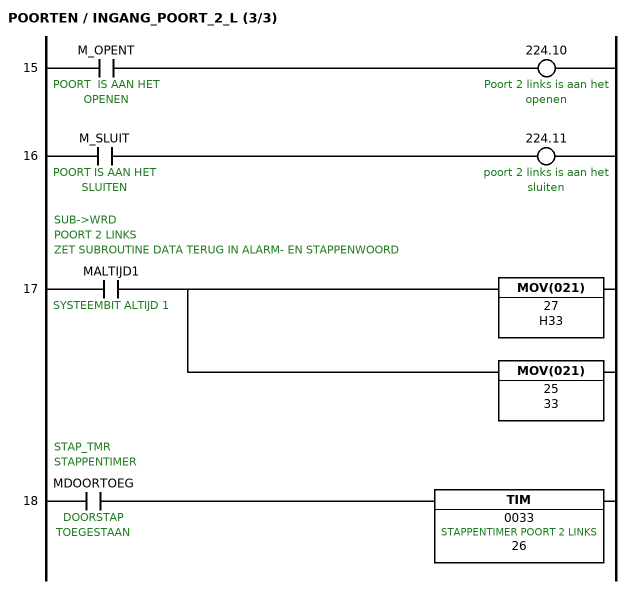
; [picture p445: POORTEN / INGANG_POORT_2_L, rungs 15-18]
; rung 15
LD M_OPENT  ; POORT  IS AAN HET OPENEN
OUT 224.10  ; Poort 2 links is aan het openen
; rung 16
LD M_SLUIT  ; POORT IS AAN HET SLUITEN
OUT 224.11  ; poort 2 links is aan het sluiten
; rung 17: SUB->WRD / POORT 2 LINKS / ZET SUBROUTINE DATA TERUG IN ALARM- EN STAPPENWOORD
LD MALTIJD1  ; SYSTEEMBIT ALTIJD 1
MOV(021) 27 H33
MOV(021) 25 33
; rung 18: STAP_TMR / STAPPENTIMER
LD MDOORTOEG  ; DOORSTAP TOEGESTAAN
TIM 0033 26  ; STAPPENTIMER POORT 2 LINKS

### Section INGANG_POORT_2_R

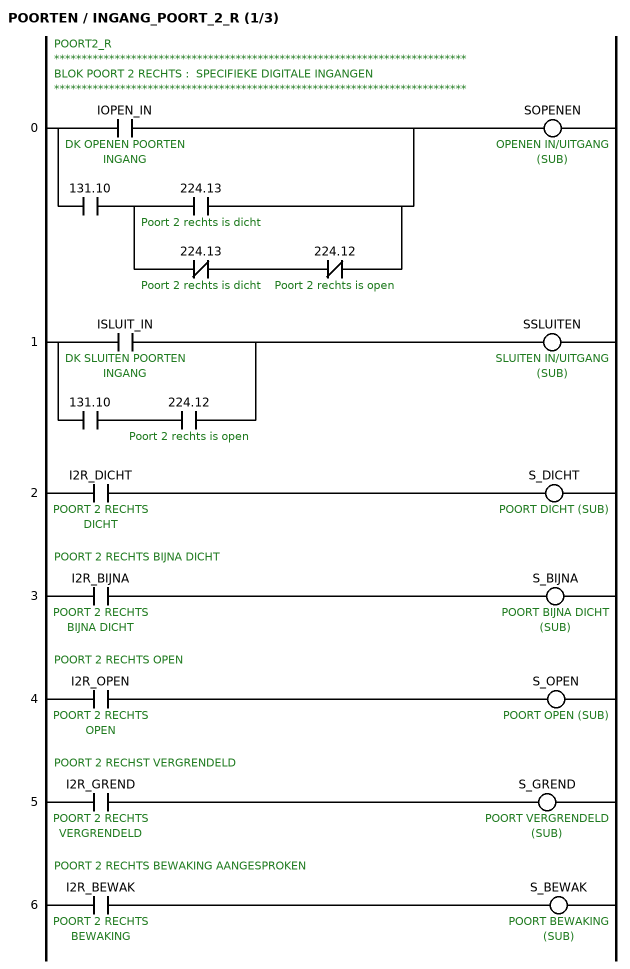
; rung 0: POORT2_R / *************************************************************************** / BLOK POORT 2 RECHTS :  SPECIFIEKE DIGITALE INGANGEN / ***************************************************************************
LD IOPEN_IN  ; DK OPENEN POORTEN INGANG
LD 131.10
LD 224.13  ; Poort 2 rechts is dicht
LDNOT 224.13  ; Poort 2 rechts is dicht
ANDNOT 224.12  ; Poort 2 rechts is open
ORLD
ANDLD
ORLD
OUT SOPENEN  ; OPENEN IN/UITGANG (SUB)
; rung 1
LD ISLUIT_IN  ; DK SLUITEN POORTEN INGANG
LD 131.10
AND 224.12  ; Poort 2 rechts is open
ORLD
OUT SSLUITEN  ; SLUITEN IN/UITGANG (SUB)
; rung 2
LD I2R_DICHT  ; POORT 2 RECHTS DICHT
OUT S_DICHT  ; POORT DICHT (SUB)
; rung 3: POORT 2 RECHTS BIJNA DICHT
LD I2R_BIJNA  ; POORT 2 RECHTS BIJNA DICHT
OUT S_BIJNA  ; POORT BIJNA DICHT (SUB)
; rung 4: POORT 2 RECHTS OPEN
LD I2R_OPEN  ; POORT 2 RECHTS OPEN
OUT S_OPEN  ; POORT OPEN (SUB)
; rung 5: POORT 2 RECHST VERGRENDELD
LD I2R_GREND  ; POORT 2 RECHTS VERGRENDELD
OUT S_GREND  ; POORT VERGRENDELD  (SUB)
; rung 6: POORT 2 RECHTS BEWAKING AANGESPROKEN
LD I2R_BEWAK  ; POORT 2 RECHTS BEWAKING
OUT S_BEWAK  ; POORT BEWAKING  (SUB)

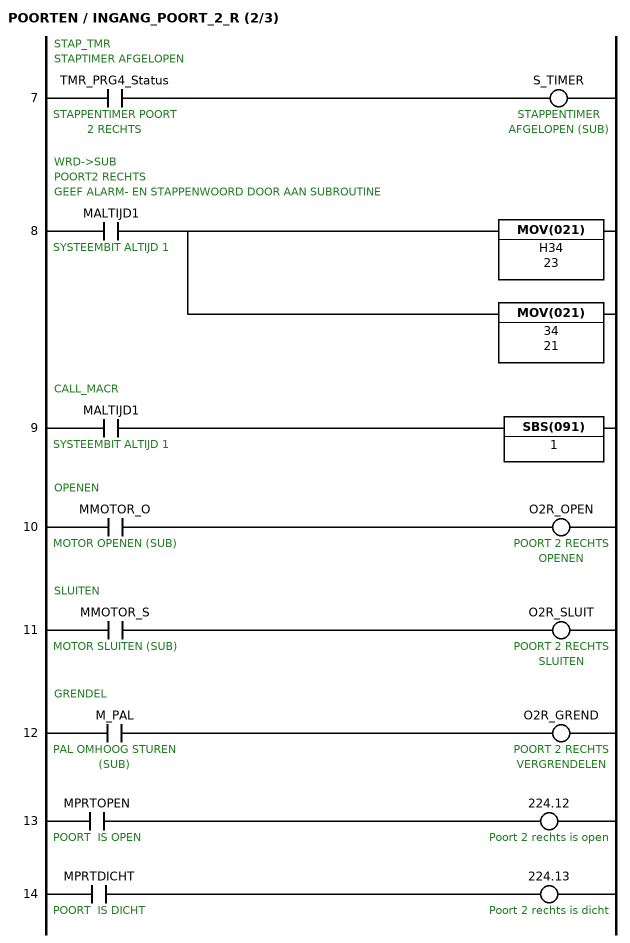
; rung 7: STAP_TMR / STAPTIMER AFGELOPEN
LD TMR_PRG4_Status  ; STAPPENTIMER POORT 2 RECHTS
OUT S_TIMER  ; STAPPENTIMER AFGELOPEN (SUB)
; rung 8: WRD->SUB / POORT2 RECHTS / GEEF ALARM- EN STAPPENWOORD DOOR AAN SUBROUTINE
LD MALTIJD1  ; SYSTEEMBIT ALTIJD 1
MOV(021) H34 23
MOV(021) 34 21
; rung 9: CALL_MACR
LD MALTIJD1  ; SYSTEEMBIT ALTIJD 1
SBS(091) 1
; rung 10: OPENEN
LD MMOTOR_O  ; MOTOR OPENEN (SUB)
OUT O2R_OPEN  ; POORT 2 RECHTS OPENEN
; rung 11: SLUITEN
LD MMOTOR_S  ; MOTOR SLUITEN (SUB)
OUT O2R_SLUIT  ; POORT 2 RECHTS SLUITEN
; rung 12: GRENDEL
LD M_PAL  ; PAL OMHOOG STUREN (SUB)
OUT O2R_GREND  ; POORT 2 RECHTS VERGRENDELEN
; rung 13
LD MPRTOPEN  ; POORT  IS OPEN
OUT 224.12  ; Poort 2 rechts is open
; rung 14
LD MPRTDICHT  ; POORT  IS DICHT
OUT 224.13  ; Poort 2 rechts is dicht

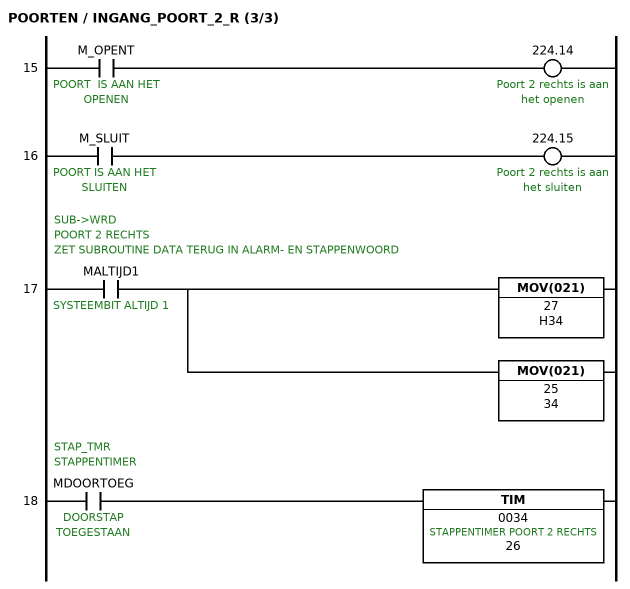
; rung 15
LD M_OPENT  ; POORT  IS AAN HET OPENEN
OUT 224.14  ; Poort 2 rechts is aan het openen
; rung 16
LD M_SLUIT  ; POORT IS AAN HET SLUITEN
OUT 224.15  ; Poort 2 rechts is aan het sluiten
; rung 17: SUB->WRD / POORT 2 RECHTS / ZET SUBROUTINE DATA TERUG IN ALARM- EN STAPPENWOORD
LD MALTIJD1  ; SYSTEEMBIT ALTIJD 1
MOV(021) 27 H34
MOV(021) 25 34
; rung 18: STAP_TMR / STAPPENTIMER
LD MDOORTOEG  ; DOORSTAP TOEGESTAAN
TIM 0034 26  ; STAPPENTIMER POORT 2 RECHTS

### Section UITGANG_POORT_3_L

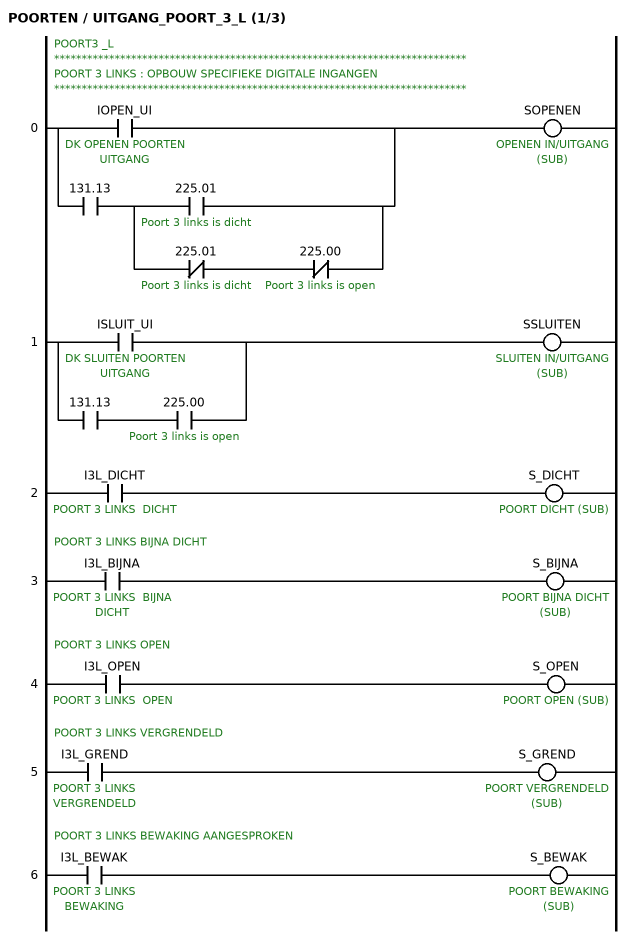
; rung 0: POORT3 _L / *************************************************************************** / POORT 3 LINKS : OPBOUW SPECIFIEKE DIGITALE INGANGEN / ***************************************************************************
LD IOPEN_UI  ; DK OPENEN POORTEN UITGANG
LD 131.13
LD 225.01  ; Poort 3 links is dicht
LDNOT 225.01  ; Poort 3 links is dicht
ANDNOT 225.00  ; Poort 3 links is open
ORLD
ANDLD
ORLD
OUT SOPENEN  ; OPENEN IN/UITGANG (SUB)
; rung 1
LD ISLUIT_UI  ; DK SLUITEN POORTEN UITGANG
LD 131.13
AND 225.00  ; Poort 3 links is open
ORLD
OUT SSLUITEN  ; SLUITEN IN/UITGANG (SUB)
; rung 2
LD I3L_DICHT  ; POORT 3 LINKS  DICHT
OUT S_DICHT  ; POORT DICHT (SUB)
; rung 3: POORT 3 LINKS BIJNA DICHT
LD I3L_BIJNA  ; POORT 3 LINKS  BIJNA DICHT
OUT S_BIJNA  ; POORT BIJNA DICHT (SUB)
; rung 4: POORT 3 LINKS OPEN
LD I3L_OPEN  ; POORT 3 LINKS  OPEN
OUT S_OPEN  ; POORT OPEN (SUB)
; rung 5: POORT 3 LINKS VERGRENDELD
LD I3L_GREND  ; POORT 3 LINKS VERGRENDELD
OUT S_GREND  ; POORT VERGRENDELD  (SUB)
; rung 6: POORT 3 LINKS BEWAKING AANGESPROKEN
LD I3L_BEWAK  ; POORT 3 LINKS BEWAKING
OUT S_BEWAK  ; POORT BEWAKING  (SUB)

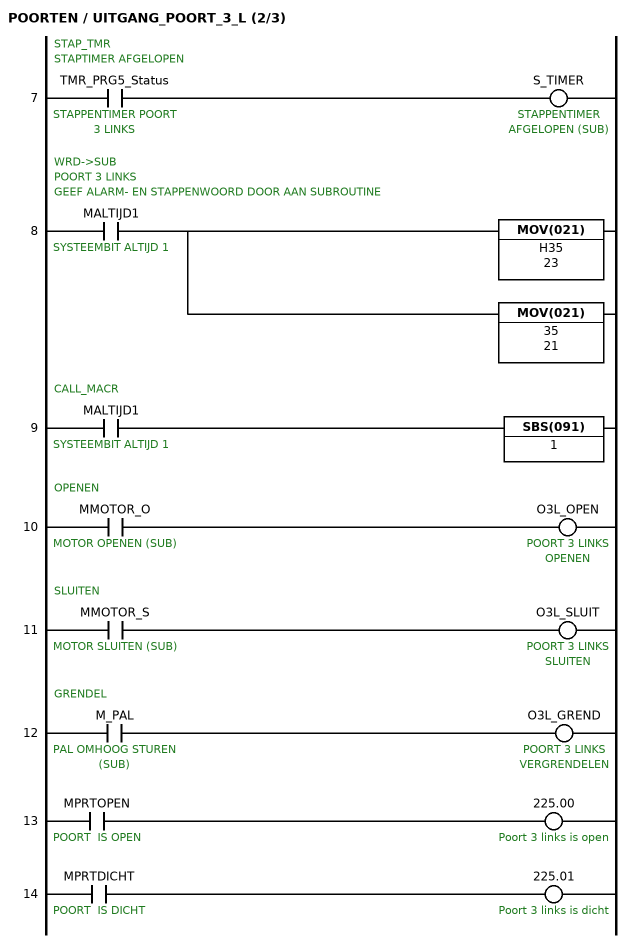
; rung 7: STAP_TMR / STAPTIMER AFGELOPEN
LD TMR_PRG5_Status  ; STAPPENTIMER POORT 3 LINKS
OUT S_TIMER  ; STAPPENTIMER AFGELOPEN (SUB)
; rung 8: WRD->SUB / POORT 3 LINKS / GEEF ALARM- EN STAPPENWOORD DOOR AAN SUBROUTINE
LD MALTIJD1  ; SYSTEEMBIT ALTIJD 1
MOV(021) H35 23
MOV(021) 35 21
; rung 9: CALL_MACR
LD MALTIJD1  ; SYSTEEMBIT ALTIJD 1
SBS(091) 1
; rung 10: OPENEN
LD MMOTOR_O  ; MOTOR OPENEN (SUB)
OUT O3L_OPEN  ; POORT 3 LINKS OPENEN
; rung 11: SLUITEN
LD MMOTOR_S  ; MOTOR SLUITEN (SUB)
OUT O3L_SLUIT  ; POORT 3 LINKS SLUITEN
; rung 12: GRENDEL
LD M_PAL  ; PAL OMHOOG STUREN (SUB)
OUT O3L_GREND  ; POORT 3 LINKS VERGRENDELEN
; rung 13
LD MPRTOPEN  ; POORT  IS OPEN
OUT 225.00  ; Poort 3 links is open
; rung 14
LD MPRTDICHT  ; POORT  IS DICHT
OUT 225.01  ; Poort 3 links is dicht

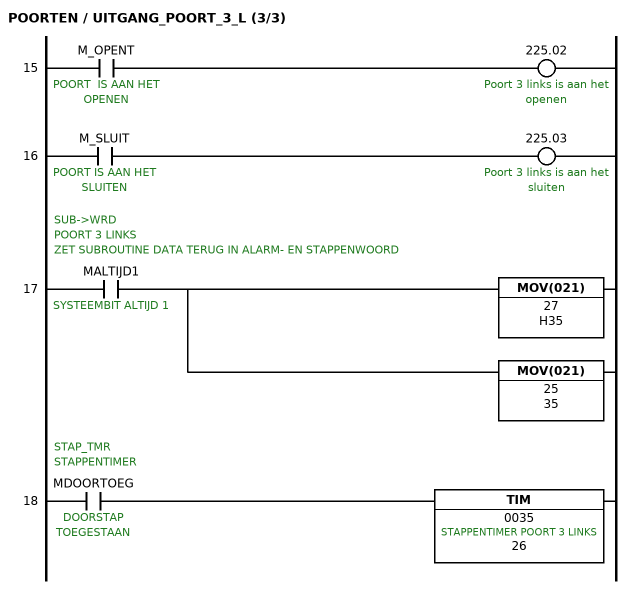
; rung 15
LD M_OPENT  ; POORT  IS AAN HET OPENEN
OUT 225.02  ; Poort 3 links is aan het openen
; rung 16
LD M_SLUIT  ; POORT IS AAN HET SLUITEN
OUT 225.03  ; Poort 3 links is aan het sluiten
; rung 17: SUB->WRD / POORT 3 LINKS / ZET SUBROUTINE DATA TERUG IN ALARM- EN STAPPENWOORD
LD MALTIJD1  ; SYSTEEMBIT ALTIJD 1
MOV(021) 27 H35
MOV(021) 25 35
; rung 18: STAP_TMR / STAPPENTIMER
LD MDOORTOEG  ; DOORSTAP TOEGESTAAN
TIM 0035 26  ; STAPPENTIMER POORT 3 LINKS

### Section UITGANG_POORT_3_R

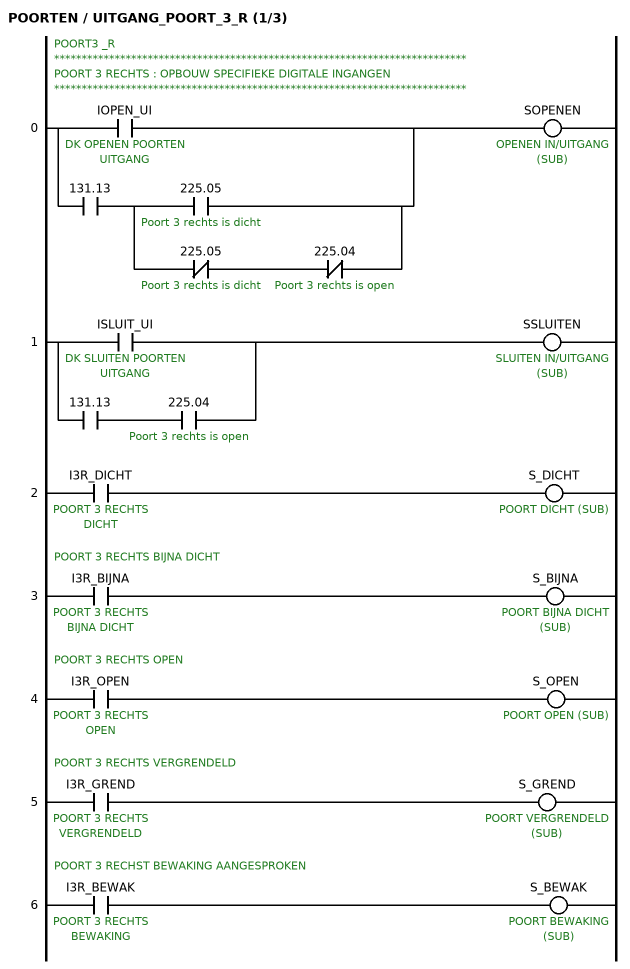
; rung 0: POORT3 _R / *************************************************************************** / POORT 3 RECHTS : OPBOUW SPECIFIEKE DIGITALE INGANGEN / ***************************************************************************
LD IOPEN_UI  ; DK OPENEN POORTEN UITGANG
LD 131.13
LD 225.05  ; Poort 3 rechts is dicht
LDNOT 225.05  ; Poort 3 rechts is dicht
ANDNOT 225.04  ; Poort 3 rechts is open
ORLD
ANDLD
ORLD
OUT SOPENEN  ; OPENEN IN/UITGANG (SUB)
; rung 1
LD ISLUIT_UI  ; DK SLUITEN POORTEN UITGANG
LD 131.13
AND 225.04  ; Poort 3 rechts is open
ORLD
OUT SSLUITEN  ; SLUITEN IN/UITGANG (SUB)
; rung 2
LD I3R_DICHT  ; POORT 3 RECHTS DICHT
OUT S_DICHT  ; POORT DICHT (SUB)
; rung 3: POORT 3 RECHTS BIJNA DICHT
LD I3R_BIJNA  ; POORT 3 RECHTS BIJNA DICHT
OUT S_BIJNA  ; POORT BIJNA DICHT (SUB)
; rung 4: POORT 3 RECHTS OPEN
LD I3R_OPEN  ; POORT 3 RECHTS OPEN
OUT S_OPEN  ; POORT OPEN (SUB)
; rung 5: POORT 3 RECHTS VERGRENDELD
LD I3R_GREND  ; POORT 3 RECHTS VERGRENDELD
OUT S_GREND  ; POORT VERGRENDELD  (SUB)
; rung 6: POORT 3 RECHST BEWAKING AANGESPROKEN
LD I3R_BEWAK  ; POORT 3 RECHTS BEWAKING
OUT S_BEWAK  ; POORT BEWAKING  (SUB)

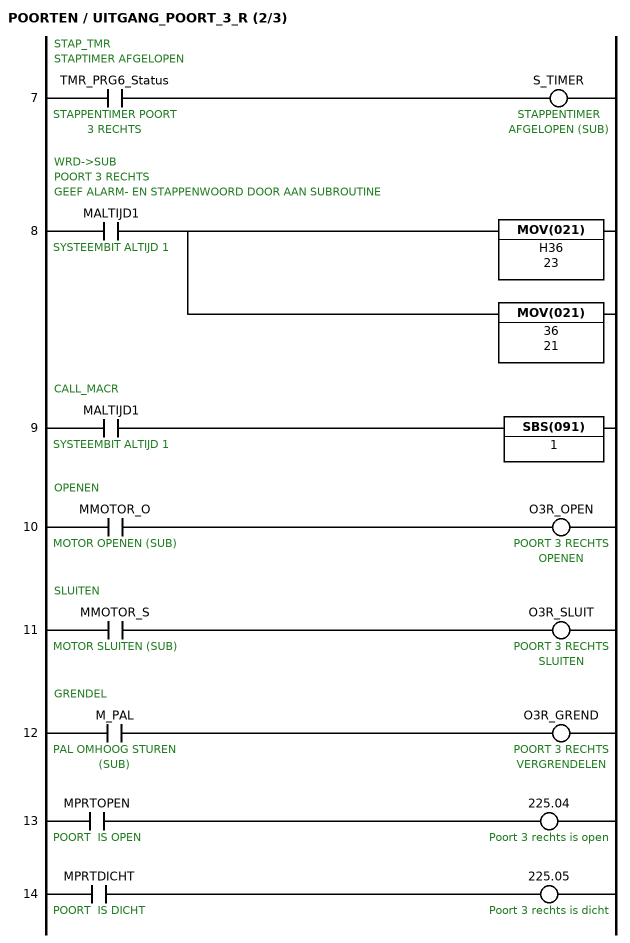
; rung 7: STAP_TMR / STAPTIMER AFGELOPEN
LD TMR_PRG6_Status  ; STAPPENTIMER POORT 3 RECHTS
OUT S_TIMER  ; STAPPENTIMER AFGELOPEN (SUB)
; rung 8: WRD->SUB / POORT 3 RECHTS / GEEF ALARM- EN STAPPENWOORD DOOR AAN SUBROUTINE
LD MALTIJD1  ; SYSTEEMBIT ALTIJD 1
MOV(021) H36 23
MOV(021) 36 21
; rung 9: CALL_MACR
LD MALTIJD1  ; SYSTEEMBIT ALTIJD 1
SBS(091) 1
; rung 10: OPENEN
LD MMOTOR_O  ; MOTOR OPENEN (SUB)
OUT O3R_OPEN  ; POORT 3 RECHTS OPENEN
; rung 11: SLUITEN
LD MMOTOR_S  ; MOTOR SLUITEN (SUB)
OUT O3R_SLUIT  ; POORT 3 RECHTS SLUITEN
; rung 12: GRENDEL
LD M_PAL  ; PAL OMHOOG STUREN (SUB)
OUT O3R_GREND  ; POORT 3 RECHTS VERGRENDELEN
; rung 13
LD MPRTOPEN  ; POORT  IS OPEN
OUT 225.04  ; Poort 3 rechts is open
; rung 14
LD MPRTDICHT  ; POORT  IS DICHT
OUT 225.05  ; Poort 3 rechts is dicht

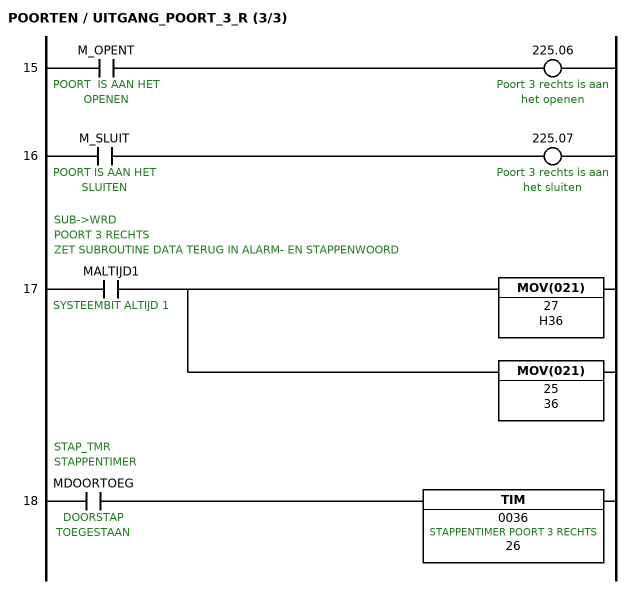
; rung 15
LD M_OPENT  ; POORT  IS AAN HET OPENEN
OUT 225.06  ; Poort 3 rechts is aan het openen
; rung 16
LD M_SLUIT  ; POORT IS AAN HET SLUITEN
OUT 225.07  ; Poort 3 rechts is aan het sluiten
; rung 17: SUB->WRD / POORT 3 RECHTS / ZET SUBROUTINE DATA TERUG IN ALARM- EN STAPPENWOORD
LD MALTIJD1  ; SYSTEEMBIT ALTIJD 1
MOV(021) 27 H36
MOV(021) 25 36
; rung 18: STAP_TMR / STAPPENTIMER
LD MDOORTOEG  ; DOORSTAP TOEGESTAAN
TIM 0036 26  ; STAPPENTIMER POORT 3 RECHTS

### Section UITGANG_POORT_4_L

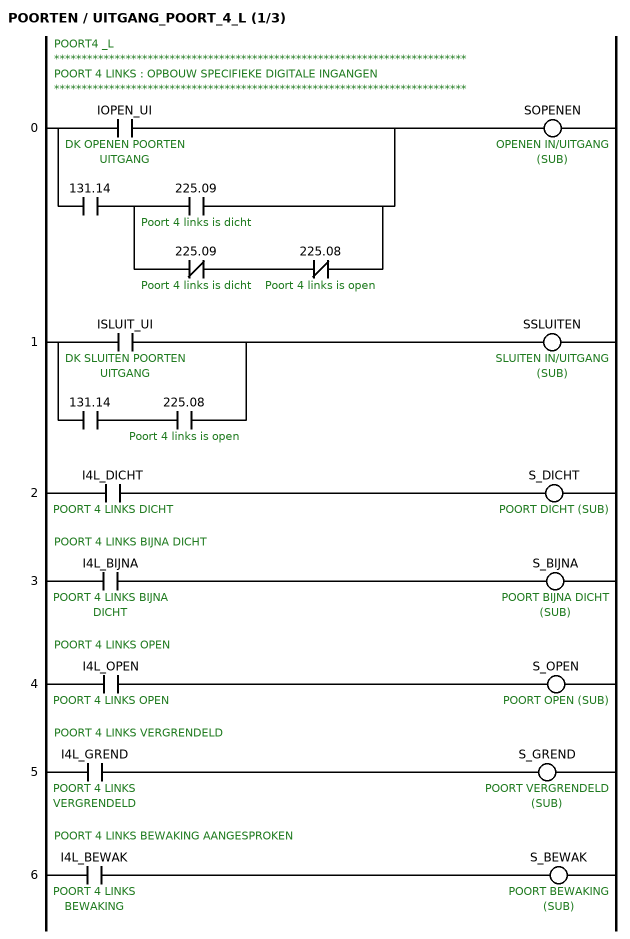
; rung 0: POORT4 _L / *************************************************************************** / POORT 4 LINKS : OPBOUW SPECIFIEKE DIGITALE INGANGEN / ***************************************************************************
LD IOPEN_UI  ; DK OPENEN POORTEN UITGANG
LD 131.14
LD 225.09  ; Poort 4 links is dicht
LDNOT 225.09  ; Poort 4 links is dicht
ANDNOT 225.08  ; Poort 4 links is open
ORLD
ANDLD
ORLD
OUT SOPENEN  ; OPENEN IN/UITGANG (SUB)
; rung 1
LD ISLUIT_UI  ; DK SLUITEN POORTEN UITGANG
LD 131.14
AND 225.08  ; Poort 4 links is open
ORLD
OUT SSLUITEN  ; SLUITEN IN/UITGANG (SUB)
; rung 2
LD I4L_DICHT  ; POORT 4 LINKS DICHT
OUT S_DICHT  ; POORT DICHT (SUB)
; rung 3: POORT 4 LINKS BIJNA DICHT
LD I4L_BIJNA  ; POORT 4 LINKS BIJNA DICHT
OUT S_BIJNA  ; POORT BIJNA DICHT (SUB)
; rung 4: POORT 4 LINKS OPEN
LD I4L_OPEN  ; POORT 4 LINKS OPEN
OUT S_OPEN  ; POORT OPEN (SUB)
; rung 5: POORT 4 LINKS VERGRENDELD
LD I4L_GREND  ; POORT 4 LINKS VERGRENDELD
OUT S_GREND  ; POORT VERGRENDELD  (SUB)
; rung 6: POORT 4 LINKS BEWAKING AANGESPROKEN
LD I4L_BEWAK  ; POORT 4 LINKS BEWAKING
OUT S_BEWAK  ; POORT BEWAKING  (SUB)

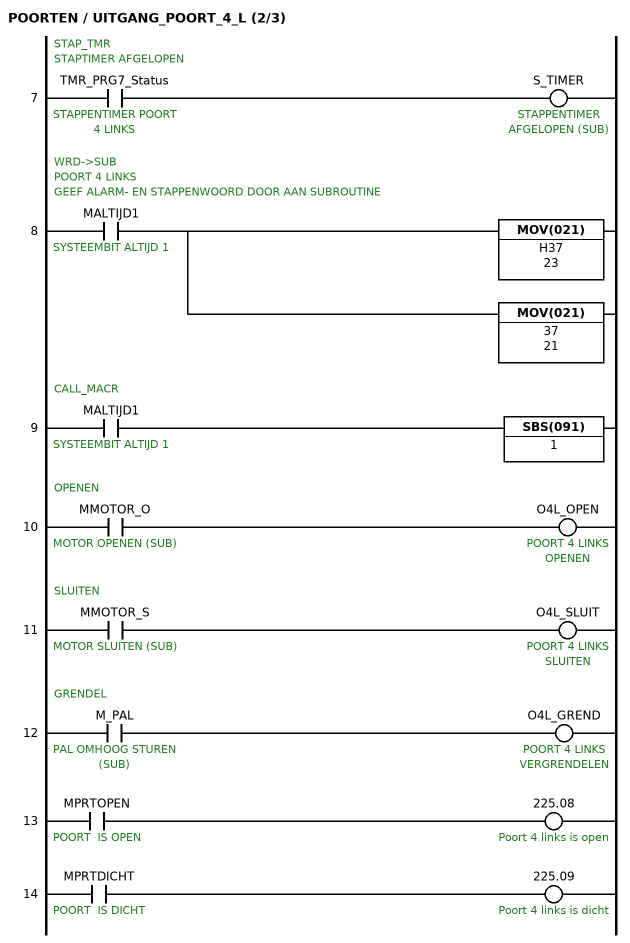
; rung 7: STAP_TMR / STAPTIMER AFGELOPEN
LD TMR_PRG7_Status  ; STAPPENTIMER POORT 4 LINKS
OUT S_TIMER  ; STAPPENTIMER AFGELOPEN (SUB)
; rung 8: WRD->SUB / POORT 4 LINKS / GEEF ALARM- EN STAPPENWOORD DOOR AAN SUBROUTINE
LD MALTIJD1  ; SYSTEEMBIT ALTIJD 1
MOV(021) H37 23
MOV(021) 37 21
; rung 9: CALL_MACR
LD MALTIJD1  ; SYSTEEMBIT ALTIJD 1
SBS(091) 1
; rung 10: OPENEN
LD MMOTOR_O  ; MOTOR OPENEN (SUB)
OUT O4L_OPEN  ; POORT 4 LINKS OPENEN
; rung 11: SLUITEN
LD MMOTOR_S  ; MOTOR SLUITEN (SUB)
OUT O4L_SLUIT  ; POORT 4 LINKS SLUITEN
; rung 12: GRENDEL
LD M_PAL  ; PAL OMHOOG STUREN (SUB)
OUT O4L_GREND  ; POORT 4 LINKS VERGRENDELEN
; rung 13
LD MPRTOPEN  ; POORT  IS OPEN
OUT 225.08  ; Poort 4 links is open
; rung 14
LD MPRTDICHT  ; POORT  IS DICHT
OUT 225.09  ; Poort 4 links is dicht

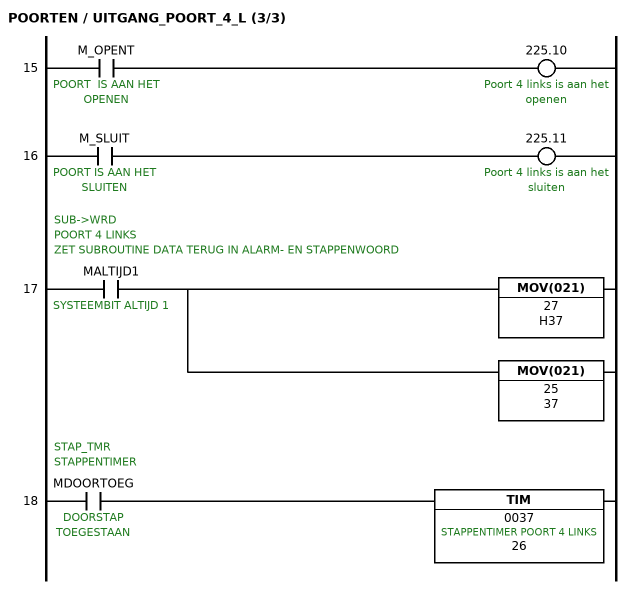
; rung 15
LD M_OPENT  ; POORT  IS AAN HET OPENEN
OUT 225.10  ; Poort 4 links is aan het openen
; rung 16
LD M_SLUIT  ; POORT IS AAN HET SLUITEN
OUT 225.11  ; Poort 4 links is aan het sluiten
; rung 17: SUB->WRD / POORT 4 LINKS / ZET SUBROUTINE DATA TERUG IN ALARM- EN STAPPENWOORD
LD MALTIJD1  ; SYSTEEMBIT ALTIJD 1
MOV(021) 27 H37
MOV(021) 25 37
; rung 18: STAP_TMR / STAPPENTIMER
LD MDOORTOEG  ; DOORSTAP TOEGESTAAN
TIM 0037 26  ; STAPPENTIMER POORT 4 LINKS

### Section UITGANG_POORT_4_R

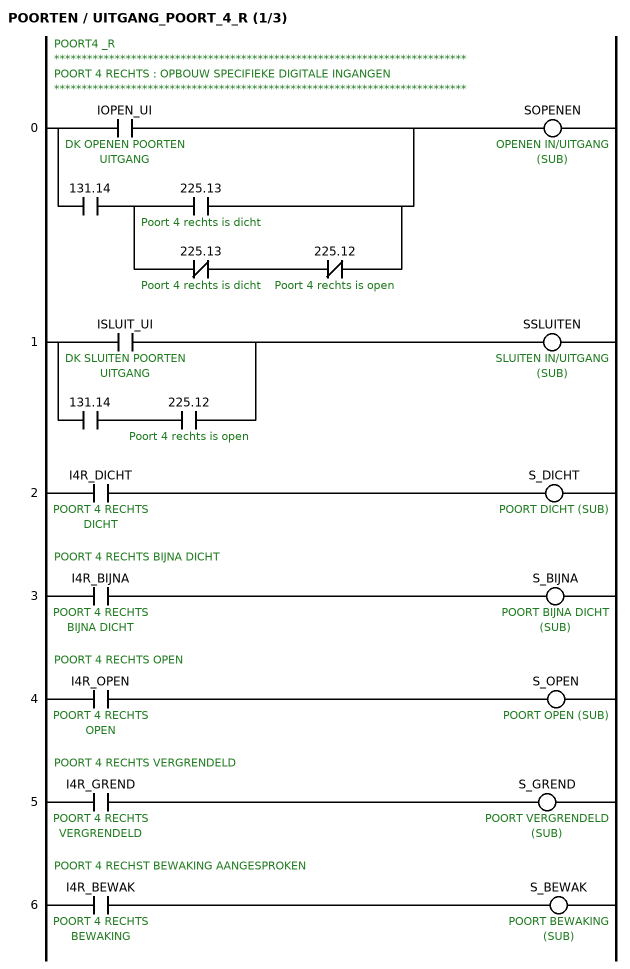
; rung 0: POORT4 _R / *************************************************************************** / POORT 4 RECHTS : OPBOUW SPECIFIEKE DIGITALE INGANGEN / ***************************************************************************
LD IOPEN_UI  ; DK OPENEN POORTEN UITGANG
LD 131.14
LD 225.13  ; Poort 4 rechts is dicht
LDNOT 225.13  ; Poort 4 rechts is dicht
ANDNOT 225.12  ; Poort 4 rechts is open
ORLD
ANDLD
ORLD
OUT SOPENEN  ; OPENEN IN/UITGANG (SUB)
; rung 1
LD ISLUIT_UI  ; DK SLUITEN POORTEN UITGANG
LD 131.14
AND 225.12  ; Poort 4 rechts is open
ORLD
OUT SSLUITEN  ; SLUITEN IN/UITGANG (SUB)
; rung 2
LD I4R_DICHT  ; POORT 4 RECHTS DICHT
OUT S_DICHT  ; POORT DICHT (SUB)
; rung 3: POORT 4 RECHTS BIJNA DICHT
LD I4R_BIJNA  ; POORT 4 RECHTS BIJNA DICHT
OUT S_BIJNA  ; POORT BIJNA DICHT (SUB)
; rung 4: POORT 4 RECHTS OPEN
LD I4R_OPEN  ; POORT 4 RECHTS OPEN
OUT S_OPEN  ; POORT OPEN (SUB)
; rung 5: POORT 4 RECHTS VERGRENDELD
LD I4R_GREND  ; POORT 4 RECHTS VERGRENDELD
OUT S_GREND  ; POORT VERGRENDELD  (SUB)
; rung 6: POORT 4 RECHST BEWAKING AANGESPROKEN
LD I4R_BEWAK  ; POORT 4 RECHTS BEWAKING
OUT S_BEWAK  ; POORT BEWAKING  (SUB)

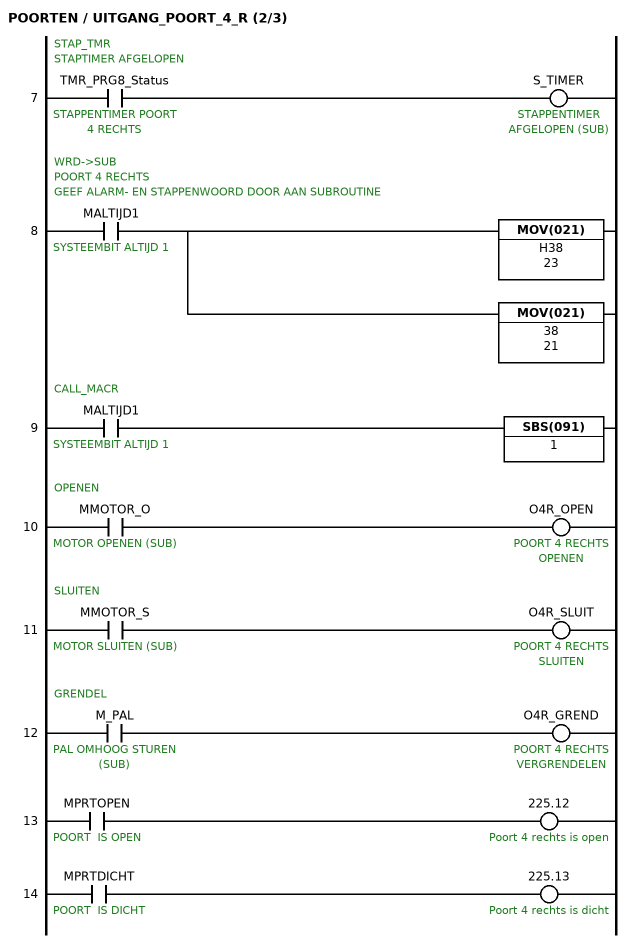
; rung 7: STAP_TMR / STAPTIMER AFGELOPEN
LD TMR_PRG8_Status  ; STAPPENTIMER POORT 4 RECHTS
OUT S_TIMER  ; STAPPENTIMER AFGELOPEN (SUB)
; rung 8: WRD->SUB / POORT 4 RECHTS / GEEF ALARM- EN STAPPENWOORD DOOR AAN SUBROUTINE
LD MALTIJD1  ; SYSTEEMBIT ALTIJD 1
MOV(021) H38 23
MOV(021) 38 21
; rung 9: CALL_MACR
LD MALTIJD1  ; SYSTEEMBIT ALTIJD 1
SBS(091) 1
; rung 10: OPENEN
LD MMOTOR_O  ; MOTOR OPENEN (SUB)
OUT O4R_OPEN  ; POORT 4 RECHTS OPENEN
; rung 11: SLUITEN
LD MMOTOR_S  ; MOTOR SLUITEN (SUB)
OUT O4R_SLUIT  ; POORT 4 RECHTS SLUITEN
; rung 12: GRENDEL
LD M_PAL  ; PAL OMHOOG STUREN (SUB)
OUT O4R_GREND  ; POORT 4 RECHTS VERGRENDELEN
; rung 13
LD MPRTOPEN  ; POORT  IS OPEN
OUT 225.12  ; Poort 4 rechts is open
; rung 14
LD MPRTDICHT  ; POORT  IS DICHT
OUT 225.13  ; Poort 4 rechts is dicht

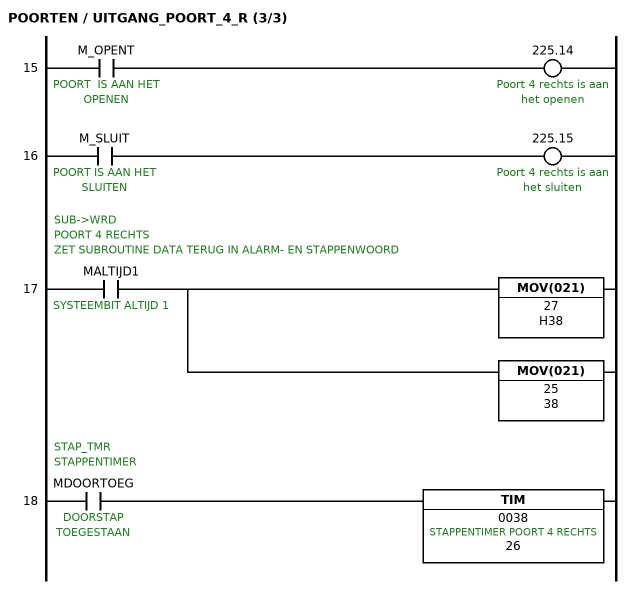
; rung 15
LD M_OPENT  ; POORT  IS AAN HET OPENEN
OUT 225.14  ; Poort 4 rechts is aan het openen
; rung 16
LD M_SLUIT  ; POORT IS AAN HET SLUITEN
OUT 225.15  ; Poort 4 rechts is aan het sluiten
; rung 17: SUB->WRD / POORT 4 RECHTS / ZET SUBROUTINE DATA TERUG IN ALARM- EN STAPPENWOORD
LD MALTIJD1  ; SYSTEEMBIT ALTIJD 1
MOV(021) 27 H38
MOV(021) 25 38
; rung 18: STAP_TMR / STAPPENTIMER
LD MDOORTOEG  ; DOORSTAP TOEGESTAAN
TIM 0038 26  ; STAPPENTIMER POORT 4 RECHTS

### Section POORTEN_ALL
; POORTEN_ALL

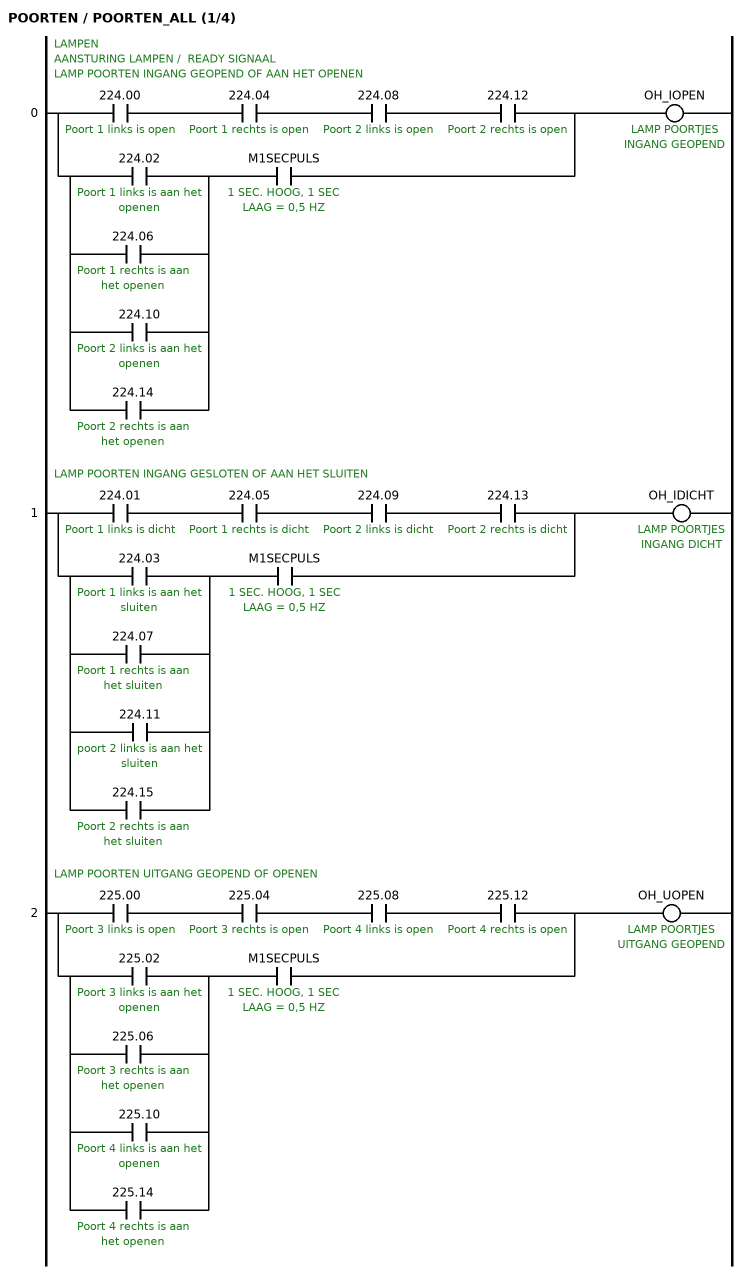
; rung 0: LAMPEN / AANSTURING LAMPEN /  READY SIGNAAL / LAMP POORTEN INGANG GEOPEND OF AAN HET OPENEN
LD 224.00  ; Poort 1 links is open
AND 224.04  ; Poort 1 rechts is open
AND 224.08  ; Poort 2 links is open
AND 224.12  ; Poort 2 rechts is open
LD 224.02  ; Poort 1 links is aan het openen
OR 224.06  ; Poort 1 rechts is aan het openen
OR 224.10  ; Poort 2 links is aan het openen
OR 224.14  ; Poort 2 rechts is aan het openen
AND M1SECPULS  ; 1 SEC. HOOG, 1 SEC LAAG = 0,5 HZ
ORLD
OUT OH_IOPEN  ; LAMP POORTJES INGANG GEOPEND
; rung 1: LAMP POORTEN INGANG GESLOTEN OF AAN HET SLUITEN
LD 224.01  ; Poort 1 links is dicht
AND 224.05  ; Poort 1 rechts is dicht
AND 224.09  ; Poort 2 links is dicht
AND 224.13  ; Poort 2 rechts is dicht
LD 224.03  ; Poort 1 links is aan het sluiten
OR 224.07  ; Poort 1 rechts is aan het sluiten
OR 224.11  ; poort 2 links is aan het sluiten
OR 224.15  ; Poort 2 rechts is aan het sluiten
AND M1SECPULS  ; 1 SEC. HOOG, 1 SEC LAAG = 0,5 HZ
ORLD
OUT OH_IDICHT  ; LAMP POORTJES INGANG DICHT
; rung 2: LAMP POORTEN UITGANG GEOPEND OF OPENEN
LD 225.00  ; Poort 3 links is open
AND 225.04  ; Poort 3 rechts is open
AND 225.08  ; Poort 4 links is open
AND 225.12  ; Poort 4 rechts is open
LD 225.02  ; Poort 3 links is aan het openen
OR 225.06  ; Poort 3 rechts is aan het openen
OR 225.10  ; Poort 4 links is aan het openen
OR 225.14  ; Poort 4 rechts is aan het openen
AND M1SECPULS  ; 1 SEC. HOOG, 1 SEC LAAG = 0,5 HZ
ORLD
OUT OH_UOPEN  ; LAMP POORTJES UITGANG GEOPEND

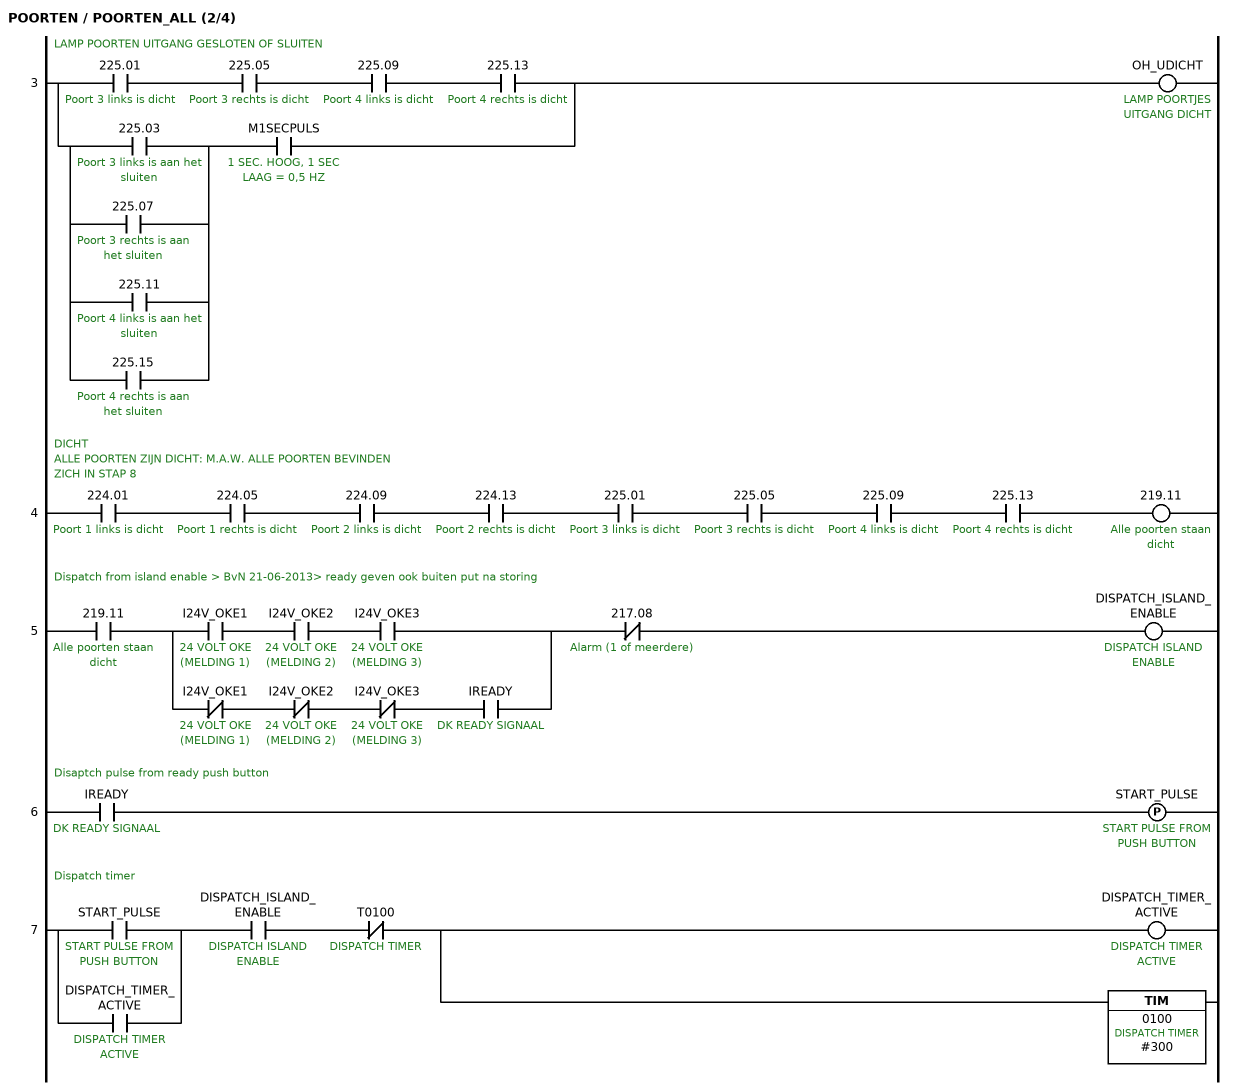
; rung 3: LAMP POORTEN UITGANG GESLOTEN OF SLUITEN
LD 225.01  ; Poort 3 links is dicht
AND 225.05  ; Poort 3 rechts is dicht
AND 225.09  ; Poort 4 links is dicht
AND 225.13  ; Poort 4 rechts is dicht
LD 225.03  ; Poort 3 links is aan het sluiten
OR 225.07  ; Poort 3 rechts is aan het sluiten
OR 225.11  ; Poort 4 links is aan het sluiten
OR 225.15  ; Poort 4 rechts is aan het sluiten
AND M1SECPULS  ; 1 SEC. HOOG, 1 SEC LAAG = 0,5 HZ
ORLD
OUT OH_UDICHT  ; LAMP POORTJES UITGANG DICHT
; rung 4: DICHT / ALLE POORTEN ZIJN DICHT: M.A.W. ALLE POORTEN BEVINDEN / ZICH IN STAP 8
LD 224.01  ; Poort 1 links is dicht
AND 224.05  ; Poort 1 rechts is dicht
AND 224.09  ; Poort 2 links is dicht
AND 224.13  ; Poort 2 rechts is dicht
AND 225.01  ; Poort 3 links is dicht
AND 225.05  ; Poort 3 rechts is dicht
AND 225.09  ; Poort 4 links is dicht
AND 225.13  ; Poort 4 rechts is dicht
OUT 219.11  ; Alle poorten staan dicht
; rung 5: Dispatch from island enable > BvN 21-06-2013> ready geven ook buiten put na storing
LD 219.11  ; Alle poorten staan dicht
LD I24V_OKE1  ; 24 VOLT OKE (MELDING 1)
AND I24V_OKE2  ; 24 VOLT OKE (MELDING 2)
AND I24V_OKE3  ; 24 VOLT OKE (MELDING 3)
LDNOT I24V_OKE1  ; 24 VOLT OKE (MELDING 1)
ANDNOT I24V_OKE2  ; 24 VOLT OKE (MELDING 2)
ANDNOT I24V_OKE3  ; 24 VOLT OKE (MELDING 3)
AND IREADY  ; DK READY SIGNAAL
ORLD
ANDLD
ANDNOT 217.08  ; Alarm (1 of meerdere)
OUT DISPATCH_ISLAND_ENABLE  ; DISPATCH ISLAND ENABLE
; rung 6: Disaptch pulse from ready push button
LD IREADY  ; DK READY SIGNAAL
DIFU(013) START_PULSE  ; START PULSE FROM PUSH BUTTON
; rung 7: Dispatch timer
LD START_PULSE  ; START PULSE FROM PUSH BUTTON
OR DISPATCH_TIMER_ACTIVE  ; DISPATCH TIMER ACTIVE
AND DISPATCH_ISLAND_ENABLE  ; DISPATCH ISLAND ENABLE
ANDNOT T0100  ; DISPATCH TIMER
OUT DISPATCH_TIMER_ACTIVE  ; DISPATCH TIMER ACTIVE
TIM 0100 #300  ; DISPATCH TIMER

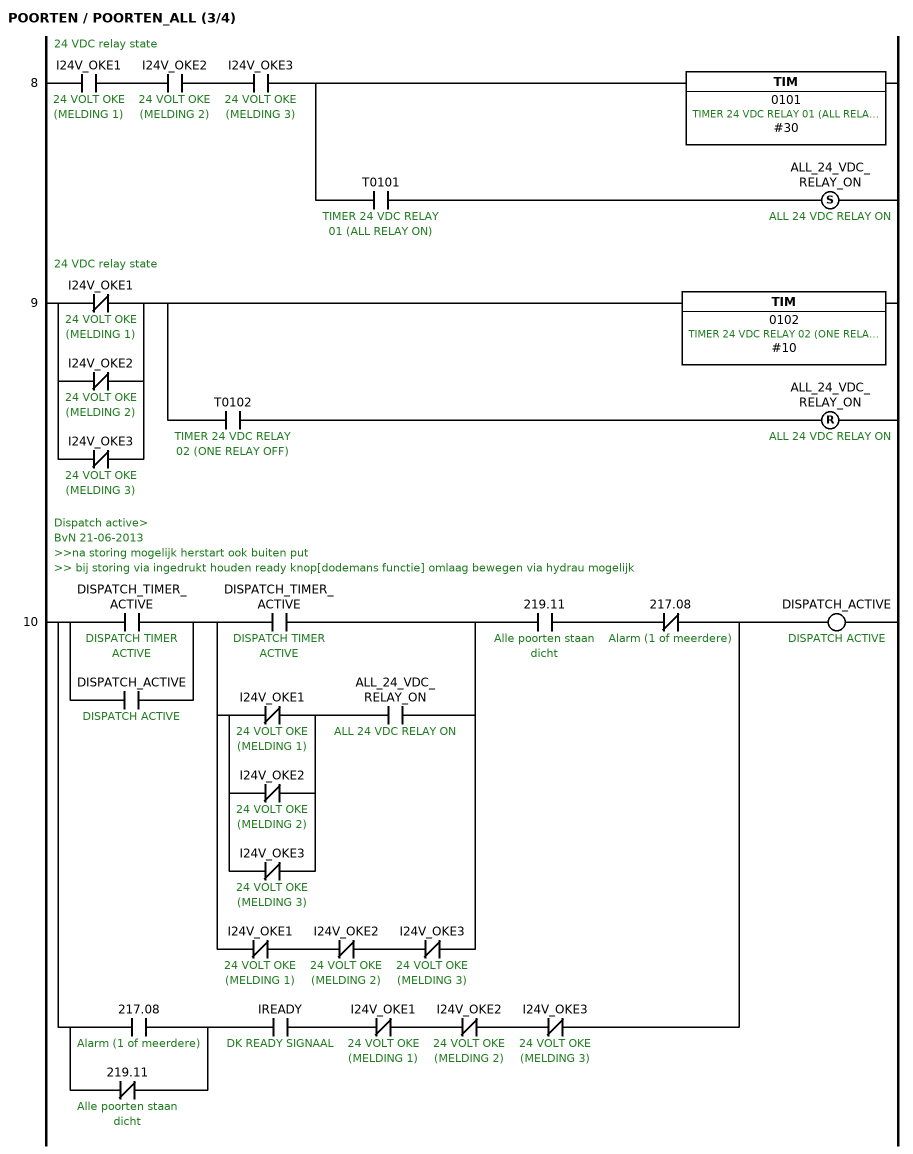
; rung 8: 24 VDC relay state
LD I24V_OKE1  ; 24 VOLT OKE (MELDING 1)
AND I24V_OKE2  ; 24 VOLT OKE (MELDING 2)
AND I24V_OKE3  ; 24 VOLT OKE (MELDING 3)
TIM 0101 #30  ; TIMER 24 VDC RELAY 01 (ALL RELAY ON)
AND T0101  ; TIMER 24 VDC RELAY 01 (ALL RELAY ON)
SET ALL_24_VDC_RELAY_ON  ; ALL 24 VDC RELAY ON
; rung 9: 24 VDC relay state
LDNOT I24V_OKE1  ; 24 VOLT OKE (MELDING 1)
ORNOT I24V_OKE2  ; 24 VOLT OKE (MELDING 2)
ORNOT I24V_OKE3  ; 24 VOLT OKE (MELDING 3)
TIM 0102 #10  ; TIMER 24 VDC RELAY 02 (ONE RELAY OFF)
AND T0102  ; TIMER 24 VDC RELAY 02 (ONE RELAY OFF)
RSET ALL_24_VDC_RELAY_ON  ; ALL 24 VDC RELAY ON
; rung 10: Dispatch active> / BvN 21-06-2013 / >>na storing mogelijk herstart ook buiten put / >> bij storing via ingedrukt houden ready knop[dodemans functie] omlaag bewegen via hydrau mogelijk
LD DISPATCH_TIMER_ACTIVE  ; DISPATCH TIMER ACTIVE
OR DISPATCH_ACTIVE  ; DISPATCH ACTIVE
LD DISPATCH_TIMER_ACTIVE  ; DISPATCH TIMER ACTIVE
LDNOT I24V_OKE1  ; 24 VOLT OKE (MELDING 1)
ORNOT I24V_OKE2  ; 24 VOLT OKE (MELDING 2)
ORNOT I24V_OKE3  ; 24 VOLT OKE (MELDING 3)
AND ALL_24_VDC_RELAY_ON  ; ALL 24 VDC RELAY ON
ORLD
LDNOT I24V_OKE1  ; 24 VOLT OKE (MELDING 1)
ANDNOT I24V_OKE2  ; 24 VOLT OKE (MELDING 2)
ANDNOT I24V_OKE3  ; 24 VOLT OKE (MELDING 3)
ORLD
ANDLD
AND 219.11  ; Alle poorten staan dicht
ANDNOT 217.08  ; Alarm (1 of meerdere)
LD 217.08  ; Alarm (1 of meerdere)
ORNOT 219.11  ; Alle poorten staan dicht
AND IREADY  ; DK READY SIGNAAL
ANDNOT I24V_OKE1  ; 24 VOLT OKE (MELDING 1)
ANDNOT I24V_OKE2  ; 24 VOLT OKE (MELDING 2)
ANDNOT I24V_OKE3  ; 24 VOLT OKE (MELDING 3)
ORLD
OUT DISPATCH_ACTIVE  ; DISPATCH ACTIVE

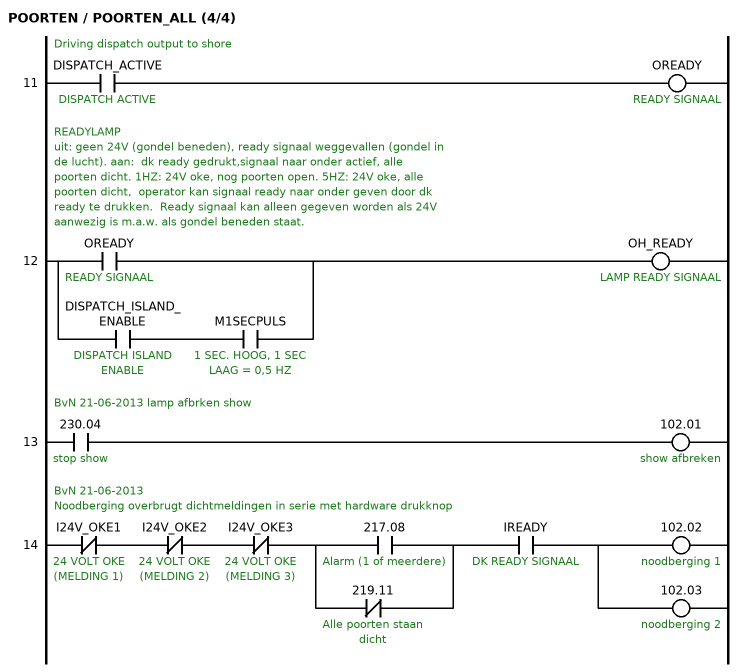
; rung 11: Driving dispatch output to shore
LD DISPATCH_ACTIVE  ; DISPATCH ACTIVE
OUT OREADY  ; READY SIGNAAL
; rung 12: READYLAMP / uit: geen 24V (gondel beneden), ready signaal weggevallen (gondel in / de lucht). aan:  dk ready gedrukt,signaal naar onder actief, alle / poorten dicht. 1HZ: 24V oke, nog poorten open. 5HZ: 24V oke, alle / poorten dicht,  operator kan signaal ready naar onder geven door dk / ready te drukken.  Ready signaal kan alleen gegeven worden als 24V / aanwezig is m.a.w. als gondel beneden staat.
LD OREADY  ; READY SIGNAAL
LD DISPATCH_ISLAND_ENABLE  ; DISPATCH ISLAND ENABLE
AND M1SECPULS  ; 1 SEC. HOOG, 1 SEC LAAG = 0,5 HZ
ORLD
OUT OH_READY  ; LAMP READY SIGNAAL
; rung 13: BvN 21-06-2013 lamp afbrken show
LD 230.04  ; stop show
OUT 102.01  ; show afbreken
; rung 14: BvN 21-06-2013 / Noodberging overbrugt dichtmeldingen in serie met hardware drukknop
LDNOT I24V_OKE1  ; 24 VOLT OKE (MELDING 1)
ANDNOT I24V_OKE2  ; 24 VOLT OKE (MELDING 2)
ANDNOT I24V_OKE3  ; 24 VOLT OKE (MELDING 3)
LD 217.08  ; Alarm (1 of meerdere)
ORNOT 219.11  ; Alle poorten staan dicht
ANDLD
AND IREADY  ; DK READY SIGNAAL
OUT 102.02  ; noodberging 1
OUT 102.03  ; noodberging 2

### Section SHOW_VERLICHTING

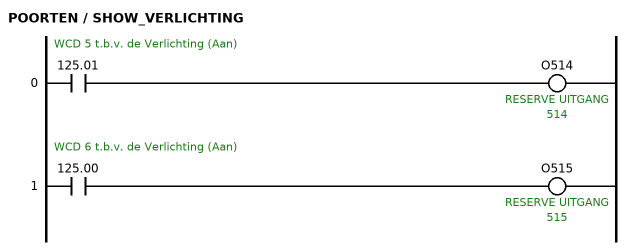
; rung 0: WCD 5 t.b.v. de Verlichting (Aan)
LD 125.01
OUT O514  ; RESERVE UITGANG 514
; rung 1: WCD 6 t.b.v. de Verlichting (Aan)
LD 125.00
OUT O515  ; RESERVE UITGANG 515

### Section SUB_DISPLAY

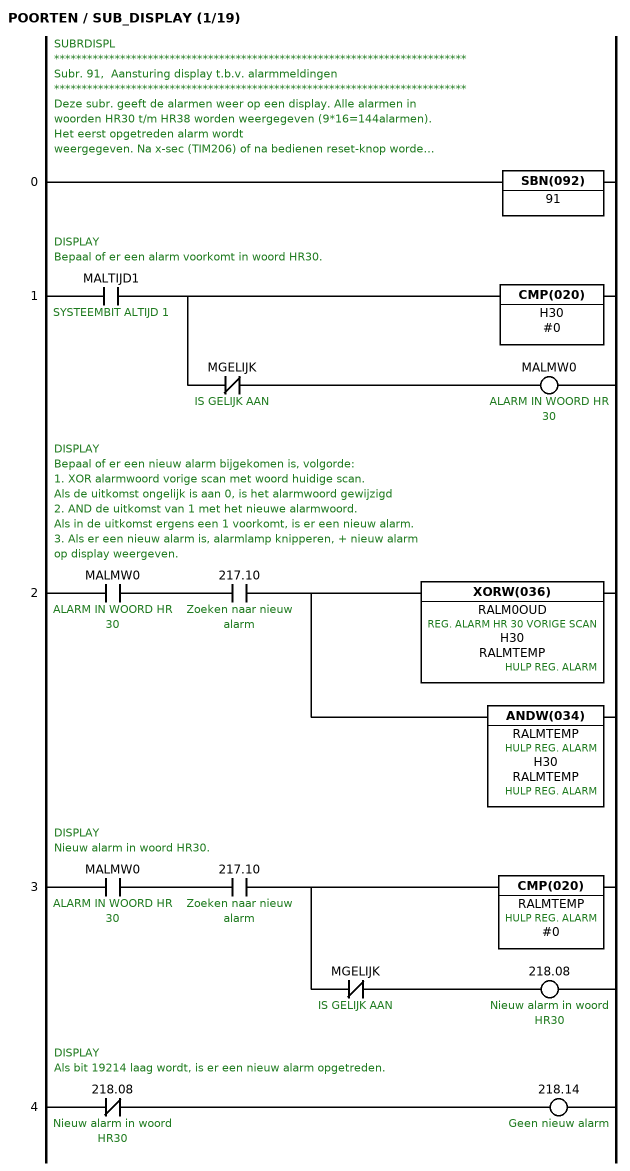
; rung 0: SUBRDISPL / *************************************************************************** / Subr. 91,  Aansturing display t.b.v. alarmmeldingen / *************************************************************************** / Deze subr. geeft de alarmen weer op een display. Alle alarmen in / woorden HR30 t/m HR38 worden weergegeven (9*16=144alarmen). / Het eerst opgetreden alarm wordt / weergegeven. Na x-sec (TIM206) of na bedienen reset-knop worden / alle alarmen gescrolld, met schroltijd TIM207. Als tijdens scrollen een / nieuw alarm optreedt, wordt dit alarm weer continu weergegeven.
SBN(092) 91
; rung 1: DISPLAY / Bepaal of er een alarm voorkomt in woord HR30.
LD MALTIJD1  ; SYSTEEMBIT ALTIJD 1
CMP(020) H30 #0
ANDNOT MGELIJK  ; IS GELIJK AAN
OUT MALMW0  ; ALARM IN WOORD HR 30
; rung 2: DISPLAY / Bepaal of er een nieuw alarm bijgekomen is, volgorde: / 1. XOR alarmwoord vorige scan met woord huidige scan. / Als de uitkomst ongelijk is aan 0, is het alarmwoord gewijzigd / 2. AND de uitkomst van 1 met het nieuwe alarmwoord. / Als in de uitkomst ergens een 1 voorkomt, is er een nieuw alarm. / 3. Als er een nieuw alarm is, alarmlamp knipperen, + nieuw alarm / op display weergeven.
LD MALMW0  ; ALARM IN WOORD HR 30
AND 217.10  ; Zoeken naar nieuw alarm
XORW(036) RALM0OUD H30 RALMTEMP  ; REG. ALARM HR 30 VORIGE SCAN, HULP REG. ALARM
ANDW(034) RALMTEMP H30 RALMTEMP  ; HULP REG. ALARM
; rung 3: DISPLAY / Nieuw alarm in woord HR30.
LD MALMW0  ; ALARM IN WOORD HR 30
AND 217.10  ; Zoeken naar nieuw alarm
CMP(020) RALMTEMP #0  ; HULP REG. ALARM
ANDNOT MGELIJK  ; IS GELIJK AAN
OUT 218.08  ; Nieuw alarm in woord HR30
; rung 4: DISPLAY / Als bit 19214 laag wordt, is er een nieuw alarm opgetreden.
LDNOT 218.08  ; Nieuw alarm in woord HR30
OUT 218.14  ; Geen nieuw alarm

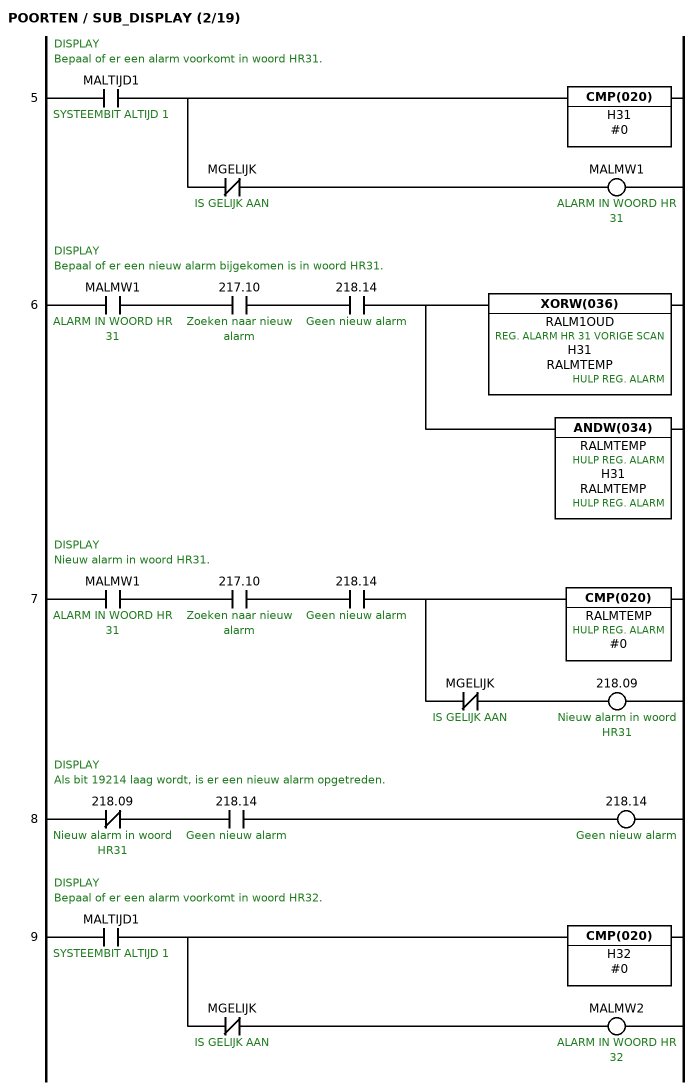
; rung 5: DISPLAY / Bepaal of er een alarm voorkomt in woord HR31.
LD MALTIJD1  ; SYSTEEMBIT ALTIJD 1
CMP(020) H31 #0
ANDNOT MGELIJK  ; IS GELIJK AAN
OUT MALMW1  ; ALARM IN WOORD HR 31
; rung 6: DISPLAY / Bepaal of er een nieuw alarm bijgekomen is in woord HR31.
LD MALMW1  ; ALARM IN WOORD HR 31
AND 217.10  ; Zoeken naar nieuw alarm
AND 218.14  ; Geen nieuw alarm
XORW(036) RALM1OUD H31 RALMTEMP  ; REG. ALARM HR 31 VORIGE SCAN, HULP REG. ALARM
ANDW(034) RALMTEMP H31 RALMTEMP  ; HULP REG. ALARM
; rung 7: DISPLAY / Nieuw alarm in woord HR31.
LD MALMW1  ; ALARM IN WOORD HR 31
AND 217.10  ; Zoeken naar nieuw alarm
AND 218.14  ; Geen nieuw alarm
CMP(020) RALMTEMP #0  ; HULP REG. ALARM
ANDNOT MGELIJK  ; IS GELIJK AAN
OUT 218.09  ; Nieuw alarm in woord HR31
; rung 8: DISPLAY / Als bit 19214 laag wordt, is er een nieuw alarm opgetreden.
LDNOT 218.09  ; Nieuw alarm in woord HR31
AND 218.14  ; Geen nieuw alarm
OUT 218.14  ; Geen nieuw alarm
; rung 9: DISPLAY / Bepaal of er een alarm voorkomt in woord HR32.
LD MALTIJD1  ; SYSTEEMBIT ALTIJD 1
CMP(020) H32 #0
ANDNOT MGELIJK  ; IS GELIJK AAN
OUT MALMW2  ; ALARM IN WOORD HR 32

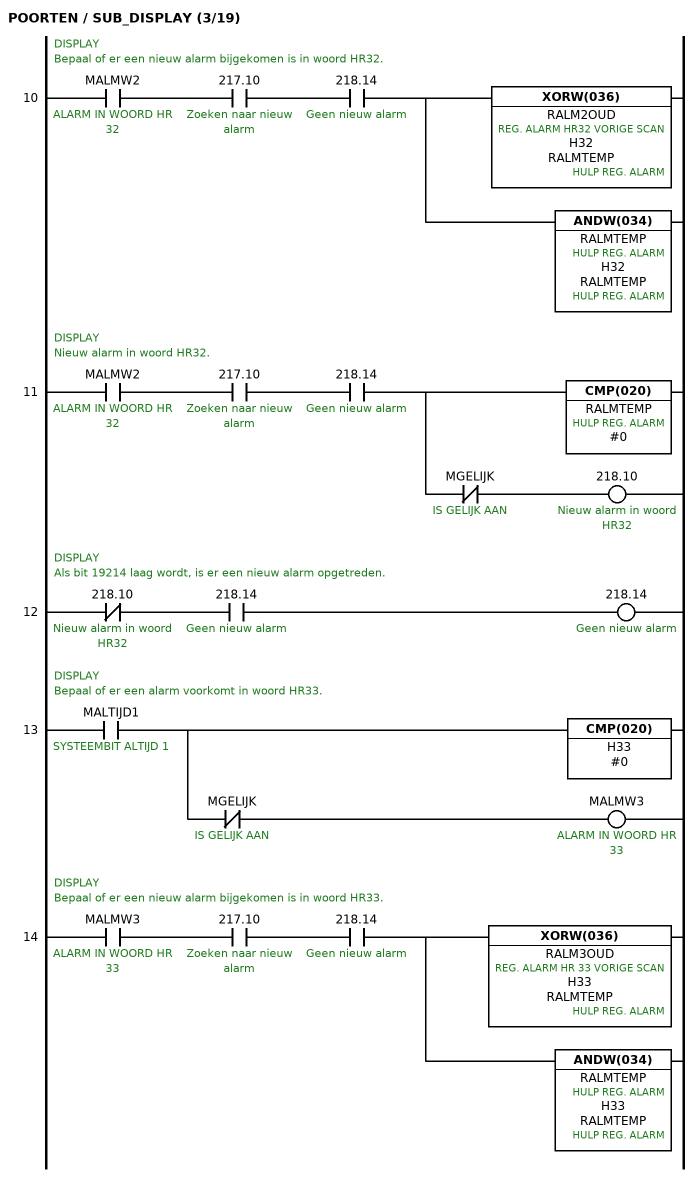
; rung 10: DISPLAY / Bepaal of er een nieuw alarm bijgekomen is in woord HR32.
LD MALMW2  ; ALARM IN WOORD HR 32
AND 217.10  ; Zoeken naar nieuw alarm
AND 218.14  ; Geen nieuw alarm
XORW(036) RALM2OUD H32 RALMTEMP  ; REG. ALARM HR32 VORIGE SCAN, HULP REG. ALARM
ANDW(034) RALMTEMP H32 RALMTEMP  ; HULP REG. ALARM
; rung 11: DISPLAY / Nieuw alarm in woord HR32.
LD MALMW2  ; ALARM IN WOORD HR 32
AND 217.10  ; Zoeken naar nieuw alarm
AND 218.14  ; Geen nieuw alarm
CMP(020) RALMTEMP #0  ; HULP REG. ALARM
ANDNOT MGELIJK  ; IS GELIJK AAN
OUT 218.10  ; Nieuw alarm in woord HR32
; rung 12: DISPLAY / Als bit 19214 laag wordt, is er een nieuw alarm opgetreden.
LDNOT 218.10  ; Nieuw alarm in woord HR32
AND 218.14  ; Geen nieuw alarm
OUT 218.14  ; Geen nieuw alarm
; rung 13: DISPLAY / Bepaal of er een alarm voorkomt in woord HR33.
LD MALTIJD1  ; SYSTEEMBIT ALTIJD 1
CMP(020) H33 #0
ANDNOT MGELIJK  ; IS GELIJK AAN
OUT MALMW3  ; ALARM IN WOORD HR 33
; rung 14: DISPLAY / Bepaal of er een nieuw alarm bijgekomen is in woord HR33.
LD MALMW3  ; ALARM IN WOORD HR 33
AND 217.10  ; Zoeken naar nieuw alarm
AND 218.14  ; Geen nieuw alarm
XORW(036) RALM3OUD H33 RALMTEMP  ; REG. ALARM HR 33 VORIGE SCAN, HULP REG. ALARM
ANDW(034) RALMTEMP H33 RALMTEMP  ; HULP REG. ALARM

